{attribute 'qualified_only'}
VAR_GLOBAL CONSTANT
	/// Fifo overhead needed to manage the string buffer
	FifoOverhead : UDINT := 10;

	/// Buffer size of temporary buffer used to persist all log messages in one cycle. 
	BufferSize : UDINT := (100 * (Tc2_System.MAX_STRING_LENGTH + FifoOverhead));
END_VAR

(* stored: Version 1.1.0.1
   GVL Constants: Id {98d3c9eb-cf89-468b-a8b6-e3b4bfd38910}, ParameterList True *)
